FUNCTION F_TwoDigits : STRING
VAR_INPUT
	x : INT;
END_VAR
VAR
	y : STRING(2);
END_VAR

// --- Simple helper: two-digit zero padding for INT -> "00".."59"
y := INT_TO_STRING(x);

IF LEN(y) = 1 THEN
	y := CONCAT('0', y); 
END_IF

F_TwoDigits := y;

END_FUNCTION

(* stored: Version 1.1.0.1, ProductVersion 3.1.4024.12
   POU F_TwoDigits: Id {6cd2584a-a696-46ac-ac87-c32672e77fae}, SpecialFunc None *)
